{attribute 'linkalways'} 
{attribute 'no_explicit_call' := 'This FB is a CLASS and must be accessed using methods or properties'}
{attribute 'enable_dynamic_creation'}
FUNCTION_BLOCK FINAL XOR_INT EXTENDS Node
VAR
	in1 : _INT(0);
	in2 : _INT(0);
	out : _INT(0);
END_VAR

METHOD PUBLIC Clone : I_Node
VAR
	pNode : POINTER TO XOR_INT;
END_VAR
pNode := __NEW(XOR_INT);
Clone := pNode^;
END_METHOD

METHOD FB_init : BOOL
VAR_INPUT
	bInitRetains : BOOL; // if TRUE, the retain variables are initialized (warm start / cold start)
	bInCopyCode : BOOL;  // if TRUE, the instance afterwards gets moved into the copy code (online change)
END_VAR
AddInput('in1',THIS^.in1);
AddInput('in2',THIS^.in2);
AddOutput('out', THIS^.out);
END_METHOD

METHOD PROTECTED OnExecute
VAR
END_VAR
out.Value := in1.Value XOR in2.Value;
END_METHOD

END_FUNCTION_BLOCK

(* stored: Version 1.1.0.1, ProductVersion 3.1.4024.15
   POU XOR_INT: Id {e73508fa-6d8d-4771-a785-dfc699963d56}, SpecialFunc None
   Folder Constructor: Id {2a7d8522-b1e5-4acd-8015-842f749db145}
   Method Clone: Id {79276ca5-07fb-4cb9-b1bf-949dc4dfa5af}
   Method FB_init: Id {2d41aee8-a2a8-41f1-96e4-c906cd4003a2}
   Method OnExecute: Id {cea7ae55-631b-481b-8801-ccdfcd16b631} *)
